// TwinCAT 3 PLC project Main_PLC_Project
// ProgramVersion: 3.1.4023.0
// libraries:
//   Tc2_SerialCom, * (Beckhoff Automation GmbH)
//   Tc2_Standard, * (Beckhoff Automation GmbH)
//   Tc2_System, * (Beckhoff Automation GmbH)
//   Tc2_Utilities, * (Beckhoff Automation GmbH)
//   Tc3_EventLogger, * (Beckhoff Automation GmbH)
//   Tc3_Module, * (Beckhoff Automation GmbH)
// project tree:
//   DUTs/ eConditionCheck.TcDUT, eControlArchitectures.TcDUT (not stored), eMainStateMachine.TcDUT, eOperationMode.TcDUT, eSensorError.TcDUT, eSystemMode.TcDUT, eXMCStateMachine.TcDUT, stOperationMode.TcDUT
//   GVLs/ AccelerationSensor.TcGVL (not stored), OperationControl.TcGVL (not stored), TEST.TcGVL, XMC.TcGVL (not stored)
//   / PlcTask.TcTTO (not stored), PlcTask_Fast.TcTTO
//   POUs/ErrorHandling/ FB_ErrorHandling.TcPOU
//   POUs/ FB_GuidanceSystem.TcPOU, FB_LevitationSystem.TcPOU, FB_ServiceModule.TcPOU, MainControl.TcPOU
//   POUs/Guidance/AccelerationSensor/ Background.TcPOU, BackgroundEL.TcPOU (not stored), FB_AccelerationSensor.TcPOU, FB_SerialCom.TcPOU
// real-time tasks:
//   TASK PlcTask: cycle T#1ms, priority 20, ADS port 351
//   TASK PlcTask_Fast: cycle T#1ms, priority 19, ADS port 350
// I/O:
//   DEVICE Gerät 1 (EtherCAT), AmsNetId 10.183.66.136.2.1
// variable links:
//   Main PLC Project/Main PLC Project Instance <-> Device 1 (EtherCAT)
//     PlcTask Inputs/TEST.iTest <-> Inputs/DevState

CONFIGURATION Main_PLC_Project
    RESOURCE PLC ON TwinCAT3
        TASK PlcTask_Fast(INTERVAL := T#1ms, PRIORITY := 19);
        PROGRAM Background WITH PlcTask_Fast : Background;
    END_RESOURCE
END_CONFIGURATION

// ---- DUTs/eConditionCheck.TcDUT
{attribute 'qualified_only'}
{attribute 'strict'}
TYPE eConditionCheck :
(
	INIT := 0,
	READY := 1,
	ERROR := 2,
	SLEEP := 3
);
END_TYPE

// ---- DUTs/eMainStateMachine.TcDUT
{attribute 'qualified_only'}
{attribute 'strict'}
TYPE eMainStateMachine :
(
	STARTUP,
	READY,
	OPERATIONAL,
	SHUTDOWN,
	ERROR
);
END_TYPE

// ---- DUTs/eOperationMode.TcDUT
{attribute 'qualified_only'}
{attribute 'strict'}
TYPE eOperationMode :
(
	RUN,
	TEST
	
);
END_TYPE

// ---- DUTs/eSensorError.TcDUT
{attribute 'qualified_only'}
{attribute 'strict'}
TYPE eSensorError :
(
	CommunicationError := 0,	
	OutOfRange := 1,
	UndefinedError := 2,
	NoError	:= 3
);
END_TYPE

// ---- DUTs/eSystemMode.TcDUT
{attribute 'qualified_only'}
{attribute 'strict'}
TYPE eSystemMode :
(
	RUN,
	SLEEP
);
END_TYPE

// ---- DUTs/eXMCStateMachine.TcDUT
{attribute 'qualified_only'}
{attribute 'strict'}
TYPE eXMCStateMachine :
(
	INIT,
	STOP,
	OP,
	ERROR
);
END_TYPE

// ---- DUTs/stOperationMode.TcDUT
TYPE stOperationMode :
STRUCT
	eMode : eOperationMode;
	bTestServiceModule : BOOL;
	bTestLevitationSystem : BOOL;
	bTestGuidanceSystem : BOOL;
	nTestMode : BYTE;
END_STRUCT
END_TYPE

// ---- GVLs/TEST.TcGVL
{attribute 'qualified_only'}
VAR_GLOBAL
	iTest AT %I* : INT;
END_VAR

// ---- POUs/Guidance/AccelerationSensor/Background.TcPOU
PROGRAM Background
VAR
END_VAR

BackgroundEL();

END_PROGRAM

// ---- POUs/ErrorHandling/FB_ErrorHandling.TcPOU
FUNCTION_BLOCK FB_ErrorHandling
VAR_INPUT
END_VAR
VAR_OUTPUT
END_VAR
VAR
END_VAR

END_FUNCTION_BLOCK

// ---- POUs/FB_GuidanceSystem.TcPOU
FUNCTION_BLOCK FB_GuidanceSystem
VAR_INPUT
END_VAR
VAR_OUTPUT
	eCondition : eConditionCheck;
END_VAR
VAR
	fbAccelerationSensor1 : FB_AccelerationSensor;
	fbAccelerationSensor2 : FB_AccelerationSensor;
	
	eMode : eSystemMode;
END_VAR

CASE eMode OF
	eSystemMode.RUN :
		fbAccelerationSensor1();
		fbAccelerationSensor2();
		
		//Condition
		IF fbAccelerationSensor1.eCondition = eConditionCheck.INIT OR fbAccelerationSensor2.eCondition = eConditionCheck.INIT THEN
			eCondition := eConditionCheck.INIT;
		ELSIF fbAccelerationSensor1.eCondition = eConditionCheck.ERROR OR fbAccelerationSensor2.eCondition = eConditionCheck.ERROR THEN
			eCondition := eConditionCheck.ERROR;
		ELSIF fbAccelerationSensor1.eCondition = eConditionCheck.READY AND fbAccelerationSensor2.eCondition = eConditionCheck.READY THEN
			eCondition := eConditionCheck.READY;
		END_IF
			
	eSystemMode.SLEEP :
		//Condition
		eCondition := eConditionCheck.SLEEP;
END_CASE

PROPERTY getAccelerationSensor1 : ARRAY [0..2] OF REAL
GET
getAccelerationSensor1 := fbAccelerationSensor1.getAcceleration;
END_GET
END_PROPERTY

PROPERTY getAccelerationSensor2 : ARRAY [0..2] OF REAL
GET
getAccelerationSensor2 := fbAccelerationSensor1.getAcceleration;
END_GET
END_PROPERTY

PROPERTY setSLEEP : BOOL
SET
VAR
	e: INT;
END_VAR
IF setSLEEP THEN
	eMode := eSystemMode.SLEEP;
ELSE
	eMode := eSystemMode.RUN;
END_IF
END_SET
END_PROPERTY

END_FUNCTION_BLOCK

// ---- POUs/Guidance/AccelerationSensor/FB_AccelerationSensor.TcPOU
FUNCTION_BLOCK FB_AccelerationSensor
VAR_INPUT
END_VAR
VAR_OUTPUT
	eCondition : eConditionCheck := eConditionCheck.INIT;
	eErrorID : eSensorError;
END_VAR
VAR
	fbEL6001	: FB_SerialCom;
	
	RxBufferPcCom	: ComBuffer;
	TxBufferPcCom	: ComBuffer;
	eComErrorID : ComError_t;
	
	acc_x : REAL;
	acc_y : REAL;	
	acc_z : REAL;
	
	fbTimer : TON;
	fbReset : TON;
	fbTrigger : R_TRIG;
	iCounter1 : UDINT;
	iCounter2 : UDINT;
	a_iPackets : ARRAY [0..9] OF UDINT;
	i : UDINT := 0;
	iSum : UDINT := 0;
	rPacketRate : REAL := 0;
	bTrigger : BOOL := FALSE;
	bCount : BOOL;
	
	fbErrorTimer : TON;
END_VAR
VAR CONSTANT
	GRAVITATIONAL_ACCELERATION : REAL := 9.81;  		//in m/s^2
END_VAR

fbEL6001(TxBuffer:=TxBufferEL, RxBuffer:=RxBufferEL, eReceiveErrorID:=eComErrorID);

acc_x := fbEL6001.getAccelerationValueX;
acc_y := fbEL6001.getAccelerationValueY;
acc_z := fbEL6001.getAccelerationValueZ;

doPacketCount();					//start packet count by setting bCount 'true' --> rPacketRate shows average rate per second

//Error
IF eComErrorID <> COMERROR_NOERROR THEN
	eErrorID := eSensorError.CommunicationError;
ELSE
	IF ABS(acc_x) > 2*GRAVITATIONAL_ACCELERATION OR ABS(acc_y) > 2*GRAVITATIONAL_ACCELERATION OR ABS(acc_z) > 2*GRAVITATIONAL_ACCELERATION THEN
		eErrorID := eSensorError.OutOfRange;
	ELSIF (ABS(acc_x) + ABS(acc_y) + ABS(acc_z)) = 0 THEN
		eErrorID := eSensorError.UndefinedError;
	ELSE
		eErrorID := eSensorError.NoError;
	END_IF
END_IF

//Condition
IF eErrorID <> eSensorError.NoError AND NOT fbErrorTimer.Q THEN
	eCondition := eConditionCheck.INIT;
	fbErrorTimer(IN := TRUE, PT := T#10S);
ELSIF eErrorID <> eSensorError.NoError AND fbErrorTimer.Q THEN
	eCondition := eConditionCheck.ERROR;
ELSIF eErrorID = eSensorError.NoError THEN
	eCondition := eConditionCheck.READY;
	fbErrorTimer.IN := FALSE;
END_IF

METHOD doPacketCount : REAL
VAR_INPUT
END_VAR
fbTimer(IN := bCount, PT := T#1S);
fbTrigger(CLK := fbTimer.IN);

IF fbTrigger.Q THEN
	iCounter1 := fbEL6001.nReceiveCounter;
END_IF

IF fbTimer.Q THEN
	iCounter2 := fbEL6001.nReceiveCounter;
	a_iPackets[i] := iCounter2 - iCounter1;
	iSum := iSum + a_iPackets[i];
	i := i + 1;
	bTrigger := TRUE;
	bCount := FALSE;
END_IF

IF i = 10 THEN
	bTrigger := FALSE;
	rPacketRate := (UDINT_TO_REAL(iSum) / UDINT_TO_REAL(i));			//times amount of packets
	i := 0;
	iSum := 0;
END_IF

fbReset(IN := bTrigger, PT := T#3S);
IF fbReset.Q THEN
	bCount := TRUE;
	bTrigger := FALSE;
END_IF
END_METHOD

PROPERTY getAcceleration : ARRAY [0..2] OF REAL
GET
getAcceleration[0] := acc_x;
getAcceleration[1] := acc_y;
getAcceleration[2] := acc_z;
END_GET
END_PROPERTY

END_FUNCTION_BLOCK

// ---- POUs/Guidance/AccelerationSensor/FB_SerialCom.TcPOU
FUNCTION_BLOCK FB_SerialCom
VAR_IN_OUT
	TxBuffer	: ComBuffer;
	RxBuffer	: ComBuffer;
	eReceiveErrorID	: ComError_t;
END_VAR
VAR
	fbReceive		: ReceiveData;
	nReceiveCounter	: UDINT;
	prefix : ARRAY[0..1] OF BYTE;
	receivedata : ARRAY [0..15] OF BYTE;
	packet_ID : BYTE := 37;
	packet_length : BYTE := 12;	
	
	crc : WORD;
	crc_check : WORD;
	pt_crc : POINTER TO WORD;
	crc12 : ARRAY [0..1] OF BYTE;	
	dataArray : ARRAY[0..11] OF BYTE;
	i : USINT;
	acc_x : ARRAY [0..3] OF BYTE;
	acc_y : ARRAY [0..3] OF BYTE;
	acc_z : ARRAY [0..3] OF BYTE;
	pt_x : POINTER TO REAL;
    x_acc : REAL;
	pt_y : POINTER TO REAL;
    y_acc : REAL;
	pt_z : POINTER TO REAL;
    z_acc : REAL;
END_VAR

prefix[0] := packet_ID;
prefix[1] := packet_length;

fbReceive(
	RXbuffer:= RxBuffer,
	pPrefix := ADR(prefix),
	LenPrefix := 2,
	pReceiveData := ADR(receivedata),
	SizeReceiveData  := 16,								
	Error=> ,
	DataReceived=>,
		);
IF fbReceive.Error <> COMERROR_NOERROR THEN
	eReceiveErrorID := fbReceive.Error;
END_IF
IF fbReceive.DataReceived THEN							
	nReceiveCounter := nReceiveCounter + 1;
END_IF

doCRC16Check1();

METHOD doCRC16Check1 : BOOL
VAR_INPUT
END_VAR
FOR i:=0 TO 11 DO
	dataArray[i] := receivedata[i+4];
END_FOR


crc := F_DATA_TO_CRC16_CCITT(
	pData := ADR(dataArray),
	cbData := BYTE_TO_UDINT(packet_length),
	crc := 16#FFFF);

crc12[0] := receivedata[2];
crc12[1] := receivedata[3];
pt_crc := ADR(crc12);
crc_check := pt_crc^;
END_METHOD

PROPERTY getAccelerationValueX : REAL
GET
IF crc_check = crc THEN

	acc_x[0] := receivedata[4];
	acc_x[1] := receivedata[5];
	acc_x[2] := receivedata[6];
	acc_x[3] := receivedata[7];
	pt_x := ADR(acc_x);
	x_acc := pt_x^;
END_IF

getAccelerationValueX := x_acc;
END_GET
END_PROPERTY

PROPERTY getAccelerationValueY : REAL
GET
IF crc_check = crc THEN
	
	acc_y[0] := receivedata[8];
	acc_y[1] := receivedata[9];
	acc_y[2] := receivedata[10];
	acc_y[3] := receivedata[11];
	pt_y := ADR(acc_y);
	y_acc := pt_y^;

END_IF
getAccelerationValueY := y_acc;
END_GET
END_PROPERTY

PROPERTY getAccelerationValueZ : REAL
GET
IF crc_check = crc THEN
	
	acc_z[0] := receivedata[12];
	acc_z[1] := receivedata[13];
	acc_z[2] := receivedata[14];
	acc_z[3] := receivedata[15];
	pt_z := ADR(acc_z);
	z_acc := pt_z^;
END_IF

getAccelerationValueZ := z_acc;
END_GET
END_PROPERTY

END_FUNCTION_BLOCK

// ---- POUs/FB_LevitationSystem.TcPOU
FUNCTION_BLOCK FB_LevitationSystem
VAR_INPUT
END_VAR
VAR_OUTPUT
	eCondition : eConditionCheck;
END_VAR
VAR
	eMode : eSystemMode;
END_VAR

PROPERTY setSLEEP : BOOL
SET
IF setSLEEP THEN
	eMode := eSystemMode.SLEEP;
ELSE
	eMode := eSystemMode.RUN;
END_IF
END_SET
END_PROPERTY

END_FUNCTION_BLOCK

// ---- POUs/FB_ServiceModule.TcPOU
FUNCTION_BLOCK FB_ServiceModule
VAR_INPUT
END_VAR
VAR_OUTPUT
	eCondition : eConditionCheck;
END_VAR
VAR
	eMode : eSystemMode;
END_VAR

PROPERTY setSLEEP : BOOL
SET
IF setSLEEP THEN
	eMode := eSystemMode.SLEEP;
ELSE
	eMode := eSystemMode.RUN;
END_IF
END_SET
END_PROPERTY

END_FUNCTION_BLOCK

// ---- POUs/MainControl.TcPOU
PROGRAM MainControl
VAR
	fbErrorHandling : FB_ErrorHandling;
	fbServiceModule : FB_ServiceModule;
	fbLevitationSystem : FB_LevitationSystem;
	fbGuidanceSystem : FB_GuidanceSystem;
	


	
	eMainState : eMainStateMachine := eMainStateMachine.STARTUP;
	fbErrorTimer : TON;										//10s
	stMode : stOperationMode;
END_VAR


CASE eMainState OF
	
	eMainStateMachine.STARTUP:
	
		IF stMode.eMode = eOperationMode.RUN THEN
			doCheckSystem();
		ELSIF stMode.eMode = eOperationMode.TEST THEN
			stMode.nTestMode.0 := stMode.bTestServiceModule;
			stMode.nTestMode.1 := stMode.bTestLevitationSystem;
			stMode.nTestMode.2 := stMode.bTestGuidanceSystem;
			
			CASE stMode.nTestMode OF
				0:
					fbServiceModule.setSLEEP := TRUE;
					fbLevitationSystem.setSLEEP := TRUE;
					fbGuidanceSystem.setSLEEP := TRUE;
				1:
					fbServiceModule.setSLEEP := FALSE;
					fbLevitationSystem.setSLEEP := TRUE;
					fbGuidanceSystem.setSLEEP := TRUE;
				2:
					fbServiceModule.setSLEEP := TRUE;
					fbLevitationSystem.setSLEEP := FALSE;
					fbGuidanceSystem.setSLEEP := TRUE;
				3:
					fbServiceModule.setSLEEP := FALSE;
					fbLevitationSystem.setSLEEP := FALSE;
					fbGuidanceSystem.setSLEEP := TRUE;
				4:
					fbServiceModule.setSLEEP := TRUE;
					fbLevitationSystem.setSLEEP := TRUE;
					fbGuidanceSystem.setSLEEP := FALSE;
				5:
					fbServiceModule.setSLEEP := FALSE;
					fbLevitationSystem.setSLEEP := TRUE;
					fbGuidanceSystem.setSLEEP := FALSE;
				6:
					fbServiceModule.setSLEEP := TRUE;
					fbLevitationSystem.setSLEEP := FALSE;
					fbGuidanceSystem.setSLEEP := FALSE;
				7:
					fbServiceModule.setSLEEP := FALSE;
					fbLevitationSystem.setSLEEP := FALSE;
					fbGuidanceSystem.setSLEEP := FALSE;
			END_CASE
			
			doCheckSystem();
		END_IF
		
		
	eMainStateMachine.READY:
		iTest := 2;

	eMainStateMachine.OPERATIONAL:
		iTest := 3;

	eMainStatemachine.SHUTDOWN:
		iTest := 4;

	eMainStateMachine.ERROR:
		iTest := 5;	




END_CASE

METHOD doCheckSystem
VAR_INPUT
END_VAR
VAR
END_VAR
fbErrorHandling();
fbServiceModule();
fbLevitationSystem();
fbGuidanceSystem();
		
IF (fbServiceModule.eCondition = eConditionCheck.READY OR fbServiceModule.eCondition = eConditionCheck.SLEEP) AND (fbLevitationSystem.eCondition = eConditionCheck.READY OR fbLevitationSystem.eCondition = eConditionCheck.SLEEP) AND (fbGuidanceSystem.eCondition = eConditionCheck.READY OR fbGuidanceSystem.eCondition = eConditionCheck.SLEEP) THEN
	eMainState := eMainStateMachine.READY;
ELSIF fbServiceModule.eCondition = eConditionCheck.ERROR OR fbLevitationSystem.eCondition = eConditionCheck.ERROR OR fbGuidanceSystem.eCondition = eConditionCheck.ERROR THEN
	fbErrorTimer(IN := TRUE, PT := T#10S);
	IF fbErrorTimer.Q THEN
		fbErrorTimer.IN := FALSE;
		eMainState := eMainStateMachine.ERROR;
	END_IF
ELSE
	fbErrorTimer.IN := FALSE;
	eMainState := eMainStateMachine.STARTUP;
END_IF
END_METHOD

END_PROGRAM
